Fanuc KAREL source: kt00333.KL

-- PROVISIONAL review KL for V770-1; original PC SHA256 72081eec14dd23584e2aa3a822c4a8e4648a49e13a7229b664b74b2dfecf3c6f
-- Incomplete behavior may be omitted. Consult companion uncertainty JSON. Do not deploy.
PROGRAM KT00333
%NOLOCKGROUP
VAR
  R1 : REAL
  I2 : INTEGER
  OUT : BOOLEAN
BEGIN
  -- UNRESOLVED_PC offsets 5-16; opcodes 2E,23
  -- UNRESOLVED_PC offsets 21-32; opcodes 2E,23
  -- UNRESOLVED_PC offsets 37-57; opcodes 21,21,64,6F,23
  -- UNRESOLVED_PC offsets 62-66; opcodes 7F
END KT00333
